(* IEC 61131-3 sources: 89152_FlorisHendrix_AfstudeerProject/89152_FlorisHendrix_ExamenProject/Stations/MachineControl/MachineControl/Class/CM_SpeedControl, 1 file *)

(* ---- CM_SpeedControl.st ---- *)
(*!
<Class
	Name               = "CM_SpeedControl"
	Revision           = "0.0"
	RealtimeTask       = "false"
	CyclicTask         = "true"
	DefCyclictime      = "10 ms"
	BackgroundTask     = "true"
	DefBackground      = "100 ms"
	Sigmatek           = "false"
	OSInterface        = "false"
	HighPriority       = "false"
	Automatic          = "false"
	UpdateMode         = "Prescan"
	SharedCommandTable = "true"
	Objectsize         = "(652,120)">
	<Channels>
		<Server Name="ClassSvr" Visualized="false" Initialize="false" WriteProtected="true" Retentive="false"/>
		<Server Name="sCycleCount" Visualized="true" Initialize="false" WriteProtected="false" Retentive="SRam"/>
		<Server Name="sDiameter" Visualized="true" Initialize="false" WriteProtected="false" Retentive="SRam"/>
		<Server Name="sMotorRunEndless" Visualized="true" Initialize="false" WriteProtected="false" Retentive="false"/>
		<Server Name="sPosInMM" Visualized="true" Initialize="false" WriteProtected="true" Retentive="false"/>
		<Server Name="sRemainingCycles" Visualized="true" Initialize="false" WriteProtected="true" Retentive="false"/>
		<Server Name="sSpeedBaseRPM" Visualized="true" Initialize="true" DefValue="36" WriteProtected="false" Retentive="SRam"/>
		<Server Name="sSpeedDegPerSec" Visualized="false" Initialize="false" WriteProtected="true" Retentive="false"/>
		<Server Name="sSpeedRPM" Visualized="true" Initialize="false" WriteProtected="true" Retentive="false"/>
		<Server Name="sStartCycles" Visualized="true" Initialize="false" WriteProtected="false" Retentive="false"/>
		<Client Name="cDI_MotorRunEndless" Required="true" Internal="false"/>
		<Client Name="cDI_ResetError" Required="true" Internal="false"/>
		<Client Name="cDI_ReverseDirection" Required="true" Internal="false"/>
		<Client Name="coLMC" Required="true" Internal="false"/>
		<Client Name="coLMCMath" Required="true" Internal="false"/>
	</Channels>
</Class>
*)
CM_SpeedControl : CLASS
  //Servers:
	ClassSvr 	: SvrChCmd_DINT;
	sSpeedBaseRPM 	: SvrCh_DINT;
	sDiameter 	: SvrCh_DINT;
	sPosInMM 	: SvrCh_DINT;
	sSpeedRPM 	: SvrCh_DINT;
	sRemainingCycles 	: SvrCh_DINT;
	sMotorRunEndless 	: SvrCh_DINT;
	sStartCycles 	: SvrCh_DINT;
	sCycleCount 	: SvrCh_DINT;
	sSpeedDegPerSec 	: SvrCh_DINT;
  //Clients:
	coLMC 	: CltChCmd__LMCAxis;
	cDI_MotorRunEndless 	: CltCh_DINT;
	cDI_ReverseDirection 	: CltCh_DINT;
	cDI_ResetError 	: CltCh_DINT;
	coLMCMath 	: CltChCmd__LMCMath_SO3;
  //Variables:
		vSetSpeed 	: DINT;
		vDegPerMM 	: DINT;
		vCircum 	: DINT;
		vPi 	: LREAL;
		vCalcSuccess 	: BOOL;
		CoS_LMCState 	: _LMCAXIS_OPMODE;
  //Functions:

	FUNCTION VIRTUAL GLOBAL Init;

	FUNCTION VIRTUAL GLOBAL CyWork
		VAR_INPUT
			EAX 	: UDINT;
		END_VAR
		VAR_OUTPUT
			state (EAX) 	: UDINT;
		END_VAR;

	FUNCTION VIRTUAL GLOBAL Background
		VAR_INPUT
			EAX 	: UDINT;
		END_VAR
		VAR_OUTPUT
			state (EAX) 	: UDINT;
		END_VAR;

	FUNCTION CalcDimensions;

	FUNCTION VIRTUAL GLOBAL sDiameter::Write
		VAR_INPUT
			input (EAX) 	: DINT;
		END_VAR
		VAR_OUTPUT
			result (EAX) 	: DINT;
		END_VAR;

	FUNCTION VIRTUAL GLOBAL sSpeedRPM::Read
		VAR_OUTPUT
			output (EAX) 	: DINT;
		END_VAR;

	FUNCTION VIRTUAL GLOBAL sStartCycles::Write
		VAR_INPUT
			input (EAX) 	: DINT;
		END_VAR
		VAR_OUTPUT
			result (EAX) 	: DINT;
		END_VAR;
  //Tables:
	FUNCTION @STD
		VAR_OUTPUT
			ret_code	: CONFSTATES;
		END_VAR;
	FUNCTION GLOBAL TAB @CT_;
END_CLASS;

#pragma usingLtd _LMCAxis
#pragma usingLtd _LMCMath_SO3

FUNCTION VIRTUAL GLOBAL CM_SpeedControl::Init
  if _FirstScan then
    coLMC.ExUnits.Write(input:=65536);
    coLMC.IntUnits.Write(360 deg);
    coLMC.Modulo.Write(360 deg);
    coLMC.VMax.Write(10 * 360 deg);
    coLMC.AMax.Write(10 * 360 deg);
    CalcDimensions(); // Bereken omtrek en graden per mm
  end_if;

  if (sSpeedBaseRPM < 10) then
    sSpeedBaseRPM.Write(10);
  end_if;

  if (sSpeedBaseRPM > 400) then
    sSpeedBaseRPM.Write(400);
  end_if;
END_FUNCTION

FUNCTION VIRTUAL GLOBAL CM_SpeedControl::CyWork
	VAR_INPUT
		EAX 	: UDINT;
	END_VAR
	VAR_OUTPUT
		state (EAX) 	: UDINT;
	END_VAR

  CoS_LMCState := coLMC;
  coLMC := coLMC.Read();

  if sStartCycles = 1 then
    cDI_MotorRunEndless := 0;
  elsif sMotorRunEndless=1 then
    cDI_MotorRunEndless := 1;
  else
    cDI_MotorRunEndless := cDI_MotorRunEndless.Read();
  end_if;

  cDI_ReverseDirection := cDI_ReverseDirection.Read();
  cDI_ResetError := cDI_ResetError.Read();

  sSpeedDegPerSec := sSpeedBaseRPM deg * 6; // 1 RPM = 6 graden/sec
  if cDI_ReverseDirection = 1 then
    sSpeedDegPerSec *= -1;
  end_if;

  vSetSpeed := coLMC.ReadVelocity(Mode:=LMCAXIS_SETVEL_APPUNIT_SEC);
  sPosInMM := coLMC.ReadPosition(LMCAXIS_SETPOS_APPUNIT)/vDegPerMM;

  case coLMC of
    PASSIVE_LMCAXIS:
      if (cDI_MotorRunEndless=1) | (sStartCycles = 1)  then
        coLMC.PowerOn(Mode:=LMCAXIS_MOVE_ANY_WAY);
      end_if;

    IDLE_LMCAXIS:
      if cDI_MotorRunEndless=1 then
        coLMC.MoveEndless(Speed:=sSpeedDegPerSec, Accel:=coLMC.AMax, Jerk:=0);
      elsif sStartCycles then
        if (sRemainingCycles > 0) then
          if (CoS_LMCState <> coLMC) then
            sRemainingCycles -= 1;
          end_if;
          coLMC.MoveRelative(
              Position:=360 deg,
              Mode:=LMCAXIS_MOVE_RELATIVE_TO_DESTINATION,
              Speed:=360 deg,
              Accel:=360 deg,
              Decel:=0,
              Jerk:=0);
        else
          sStartCycles := 0;
        end_if;
      else
        coLMC.PowerOff(Mode:=LMCAXIS_SMOOTH_STOPP);
      end_if;

    MOVE_LMCAXIS:
      if (cDI_MotorRunEndless=1) then
        if (vSetSpeed <> sSpeedDegPerSec) then
          if (vSetSpeed >= 0) XOR (sSpeedDegPerSec>=0) then
            coLMC.StopMove(Decel:=coLMC.AMax, Jerk:=0); // Richtingsverandering
          else
            coLMC.MoveEndless(Speed:=sSpeedDegPerSec, Accel:=coLMC.AMax, Jerk:=0);
          end_if;
        end_if;
      elsif (sStartCycles = 0) then
        coLMC.StopMove(Decel:=coLMC.AMax, Jerk:=0);
      end_if;
  end_case;

	state := READY;
END_FUNCTION

FUNCTION VIRTUAL GLOBAL CM_SpeedControl::Background
	VAR_INPUT
		EAX 	: UDINT;
	END_VAR
	VAR_OUTPUT
		state (EAX) 	: UDINT;
	END_VAR

	state := READY;
END_FUNCTION

FUNCTION CM_SpeedControl::CalcDimensions
  if sDiameter<=0 then
    sDiameter.Write(200);
  end_if;

  vPi := 4 * coLMCMath.atan2(1,1,#vCalcSuccess); // p-berekening via atan2
  vCircum := to_Dint(sDiameter * vPi);
  vDegPerMM := 360 deg / vCircum;
END_FUNCTION

FUNCTION VIRTUAL GLOBAL CM_SpeedControl::sDiameter::Write
	VAR_INPUT
		input (EAX) 	: DINT;
	END_VAR
	VAR_OUTPUT
		result (EAX) 	: DINT;
	END_VAR

	sDiameter := input;
	result := sDiameter;
  CalcDimensions(); // Herbereken bij nieuwe diameter
END_FUNCTION

FUNCTION VIRTUAL GLOBAL CM_SpeedControl::sSpeedRPM::Read
	VAR_OUTPUT
		output (EAX) 	: DINT;
	END_VAR

  sSpeedRPM:= 60 * vSetSpeed / (360 deg); // Omrekening van deg/sec naar RPM
	output := sSpeedRPM;
END_FUNCTION

FUNCTION VIRTUAL GLOBAL CM_SpeedControl::sStartCycles::Write
	VAR_INPUT
		input (EAX) 	: DINT;
	END_VAR
	VAR_OUTPUT
		result (EAX) 	: DINT;
	END_VAR

	sStartCycles := input;
  if sStartCycles = 1 then
    sRemainingCycles := sCycleCount;
  end_if;
	result := sStartCycles;
END_FUNCTION
